// TIA Portal V17 export
// export: Created 2025-01-08T13:55:32.170773Z, ExportSetting WithDefaults, DisplayName Totally Integrated Automation Portal, DisplayVersion V17, DisplayName TIA Portal Openness, DisplayVersion V17, DisplayName TIA Portal Version Control Interface, DisplayVersion V17, DisplayName SINAMICS Startdrive Advanced, DisplayVersion V17 Update2, DisplayName SINAMICS Startdrive G130, G150, S120, S150, SINAMICS MV, S210, DisplayVersion V17 Update2, DisplayName SINAMICS Startdrive G110M, G120, G120C, G120D, G120P, G115D, DisplayVersion V17 Update2, DisplayName STEP 7 Professional, DisplayVersion V17, DisplayName STEP 7 Safety, DisplayVersion V17, DisplayName WinCC Advanced, DisplayVersion V17
DATA_BLOCK "DB - 05_Alarms_From_HSM"   // DB550
{ S7_Optimized_Access := 'FALSE' }
VERSION : 0.1
// stored: AutoNumber false, DBAccessibleFromOPCUA true, DBAccessibleFromWebserver true, IsOnlyStoredInLoadMemory false, IsWriteProtectedInAS false
   VAR
      HSM1 : "HSM_AlarmWarning";
      HSM2 : "HSM_AlarmWarning";
      HSM3 : "HSM_AlarmWarning";
      iWarning00_From_HSM_X : Int;
      iWarning01_From_HSM_X : Int;
      iWarning02_From_HSM_X : Int;
      iWarning03_From_HSM_X : Int;
      iWarning04_From_HSM_X : Int;
      iWarning05_From_HSM_X : Int;
      iWarning06_From_HSM_X : Int;
      iWarning07_From_HSM_X : Int;
      iWarning08_From_HSM_X : Int;
      iWarning09_From_HSM_X : Int;
      iWarning10_From_HSM_X : Int;
      iWarning11_From_HSM_X : Int;
      iWarning12_From_HSM_X : Int;
      iWarning13_From_HSM_X : Int;
      iWarning14_From_HSM_X : Int;
      iWarning15_From_HSM_X : Int;
      iError00_From_HSM_X : Int;
      iError01_From_HSM_X : Int;
      iError02_From_HSM_X : Int;
      iError03_From_HSM_X : Int;
      iError04_From_HSM_X : Int;
      iError05_From_HSM_X : Int;
      iError06_From_HSM_X : Int;
      iError07_From_HSM_X : Int;
      iError08_From_HSM_X : Int;
      iError09_From_HSM_X : Int;
      iError10_From_HSM_X : Int;
      iError11_From_HSM_X : Int;
      iError12_From_HSM_X : Int;
      iError13_From_HSM_X : Int;
      iError14_From_HSM_X : Int;
      iError15_From_HSM_X : Int;
   END_VAR
BEGIN
END_DATA_BLOCK
